// TIA Portal V20 export
// export: Created 2026-07-10T11:12:33.8983641Z, ExportSetting WithDefaults, DisplayName Totally Integrated Automation Portal, DisplayVersion V20, DisplayName TIA Portal Openness, DisplayVersion V20, DisplayName TIA Portal Version Control Interface, DisplayVersion V20, DisplayName STEP 7 Professional, DisplayVersion V20, DisplayName STEP 7 Safety, DisplayVersion V20, DisplayName WinCC Basic/Comfort/Advanced, DisplayVersion V20, DisplayName WinCC Unified, DisplayVersion V20
FUNCTION_BLOCK "StepGenerator"   // FB22, SCL
{ S7_Optimized_Access := 'TRUE' }
VERSION : 0.1
// stored: AutoNumber true, IsIECCheckEnabled false, IsRetainMemResEnabled false, MemoryReserve 100, SetENOAutomatically false, UDAEnableTagReadback false
   VAR_INPUT
      Enable : Bool;
      Tanklevel : Real;
      TankLevelSetpoint : Real;
      KP : Real := 2.0;
      KI : Real := 0.2;
      KD : Real := 0.5;
      TI : Time := T#1s;
      LimitMin : Real := -100.0;
      LimitMax : Real := 100.0;
      DeadZone : Real := 1.0;
   END_VAR
   VAR_OUTPUT
      DamperPosition : Real;
   END_VAR
   VAR
      "e" : Real;
      PValue : Real;
      IValue : Real;
      DValue : Real;
      init : Bool;
      TopLevelSetPoint : Real;
      BottomlevelSetPoint : Real;
      PrevValue : Real;
      TON1 { S7_SetPoint := 'True'} : TON_TIME;
   END_VAR
BEGIN
   IF NOT #Enable THEN
       #init := false;
       #IValue := 0;
       #DValue := 0;
   END_IF;

   #TopLevelSetPoint := #TankLevelSetpoint + #DeadZone;
   #BottomlevelSetPoint := #TankLevelSetpoint - #DeadZone;

   #TON1(IN:=TRUE,
         PT:=#TI);



   IF #TON1.Q THEN
       IF #Tanklevel > #TopLevelSetPoint THEN
           #e := #e - #KP;
       ELSIF #Tanklevel < #BottomlevelSetPoint THEN
           #e := #e + #KP;
       END_IF;
       #DamperPosition := #e;
       RESET_TIMER(#TON1);
   END_IF;
END_FUNCTION_BLOCK
